(* IEC 61131-3 sources: crb-codesys/generation/scripts/repoeval/重型运输系统/core/FUN, 14 files *)

(* ---- percentCalc.st ---- *)
FUNCTION percentCalc : REAL
VAR_INPUT
	level		:INT;	//1->地轨	2->天轨
	idx			:INT;	//挡板索引编号
END_VAR
VAR
	c			:REAL;
	p			:REAL;
END_VAR

//伸出百分比计算
CASE level OF
	1:
		IF gDev.grd[idx].sensor.position < 3 THEN
			RETURN;
		END_IF
		c := gDev.grd[idx].sensor.position - gDev.grd[idx].sensor.retractVal;
		p := gDev.grd[idx].sensor.extendVal - gDev.grd[idx].sensor.retractVal;
		percentCalc := c * 100 / p;
	2:
		IF gDev.sky[idx].sensor.position < 3 THEN
			RETURN;
		END_IF
		c := gDev.sky[idx].sensor.position - gDev.sky[idx].sensor.retractVal;
		p := gDev.sky[idx].sensor.extendVal - gDev.sky[idx].sensor.retractVal;
		percentCalc := c * 100 / p;
END_CASE

(* ---- setButtonByDirect.st ---- *)
FUNCTION setButtonByDirect : BOOL
VAR_INPUT
	level		:INT;	//1->地轨	2->天轨
	idx			:INT;	//挡板索引编号
	direct		:TargetDirect;
END_VAR
VAR
END_VAR
//	本函数用于根据输入参数 操作UI界面的按钮变量
CASE level OF
	1:
		IF idx = 0 OR idx > 10 THEN		//参数校验
			RETURN;
		END_IF
		CASE direct OF
			TargetDirect.extend:
				gUI.grd[idx].btnStop := FALSE;
				gUI.grd[idx].btnExtend := TRUE;
				gUI.grd[idx].btnRetract := FALSE;
			TargetDirect.retract:
				gUI.grd[idx].btnStop := FALSE;
				gUI.grd[idx].btnExtend := FALSE;
				gUI.grd[idx].btnRetract := TRUE;
			TargetDirect.stop:
				gUI.grd[idx].btnStop := FALSE;
				gUI.grd[idx].btnExtend := FALSE;
				gUI.grd[idx].btnRetract := FALSE;
		END_CASE
	2:
		IF idx > 10 THEN		//参数校验
			RETURN;
		END_IF
		CASE direct OF
			TargetDirect.extend:
				gUI.sky[idx].btnStop := FALSE;
				gUI.sky[idx].btnExtend := TRUE;
				gUI.sky[idx].btnRetract := FALSE;
			TargetDirect.retract:
				gUI.sky[idx].btnStop := FALSE;
				gUI.sky[idx].btnExtend := FALSE;
				gUI.sky[idx].btnRetract := TRUE;
			TargetDirect.stop:
				gUI.sky[idx].btnStop := FALSE;
				gUI.sky[idx].btnExtend := FALSE;
				gUI.sky[idx].btnRetract := FALSE;
		END_CASE

END_CASE;

(* ---- updateDevStatus.st ---- *)
FUNCTION updateDevStatus : DevStatus
VAR_INPUT
	level		:INT;		//1->地轨	2->天轨
	idx			:INT;		//挡板索引编号
	errorVal	:REAL;		//误差范围
END_VAR
VAR
	extendVal	:REAL;		//伸出值
	retractVal	:REAL;		//缩回到位值
	nowVal		:REAL;		//当前值
	stat		:DevStatus;	//设备状态
END_VAR

(* 本函数用于根据设备的标定伸出/缩回值以及当前位置
** 判断该缸体是否处于伸出/缩回到位状态，如果到位更新参数
*)

stat := DevStatus.unknown;	//初始化状态量
CASE level OF
	1:
		extendVal := gDev.grd[idx].sensor.extendVal;
		retractVal := gDev.grd[idx].sensor.retractVal;
		nowVal := gDev.grd[idx].sensor.position;
		stat := gDev.grd[idx].state;
	2:
		extendVal := gDev.sky[idx].sensor.extendVal;
		retractVal := gDev.sky[idx].sensor.retractVal;
		nowVal := gDev.sky[idx].sensor.position;
		stat := gDev.sky[idx].state;
END_CASE

IF nowVal > 1 THEN
	IF nowVal < retractVal + errorVal THEN
		stat := DevStatus.retracted;
	ELSIF nowVal > extendVal - errorVal THEN
		stat := DevStatus.extended;
	ELSE
		IF stat <> DevStatus.runing THEN
			stat := DevStatus.error;
		END_IF
	END_IF
ELSE
	stat := DevStatus.unknown;
END_IF

CASE level OF
	1:
		gDev.grd[idx].state := stat;
	2:
		gDev.sky[idx].state := stat;
END_CASE

updateDevStatus := stat;

(* ---- BasePIDCtrl.st ---- *)
FUNCTION_BLOCK BasePIDCtrl
VAR_INPUT
	Act_Val 	:REAL;			//实际值
	Set_Val		:REAL;			//设定值
	Kp			:REAL;
	Ki			:REAL;
	Kd			:REAL;
	Y_MAX		:REAL;
	Y_MIN		:REAL;
	rCycle		:REAL;			//单位/s
	Reset		:BOOL;
END_VAR
VAR_OUTPUT
	Y			:REAL;
	LimitActive	:BOOL;
END_VAR
VAR
	fCycle			:REAL;
	CycleTime		:TIME ;
	Err				:REAL;    		//本次误差
	LastErr			:REAL;    		//上次误差
	KiErrSum		:REAL;			//积分累计误差
	KdErr			:REAL;			//微分误差
	Result			:REAL;			//计算结果
	Result_OUT		:REAL;		    //限制结果
	trig			:R_TRIG ;
	ton				:TON ;
END_VAR

IF  rCycle < 0.01 THEN  //10ms最小
	fCycle := 0.01;
ELSE
	fCycle := rCycle;
END_IF

CycleTime := REAL_TO_TIME (TIME_TO_REAL(T#1S) * fCycle);
ton (IN := NOT ton.Q ,PT := CycleTime ,Q =>);
trig (CLK := ton.Q  ,Q =>);

IF trig.Q THEN 			//PID计算
	Err := Set_Val - Act_Val;  //误差计算
	KiErrSum := KiErrSum + Err ;   //积分计算
	KdErr := Err -LastErr;    //微分计算
	LastErr := Err;
	(*IF ABS(Err) < 10 THEN		//误差较低时才开启积分
		KiErrSum := KiErrSum + Err ;   //积分计算
	END_IF*)
	Result :=  Kp * Err + Ki * KiErrSum + Kd * KdErr;
END_IF

IF Result > Y_MAX  THEN         //限幅度输出
	Result_OUT := Y_MAX ;
	LimitActive := TRUE ;
ELSIF Result < Y_MIN THEN
	Result_OUT := Y_MIN  ;
	LimitActive := TRUE ;
ELSE
	Result_OUT := Result ;
	LimitActive :=FALSE ;
END_IF
IF Reset THEN   //pid 不输出
	KiErrSum := 0;
	KdErr := 0;
	LastErr	:= 0;
	Y := 0;
ELSE
	Y := Result_OUT;
END_IF

(* ---- CommandExecutor.st ---- *)
FUNCTION_BLOCK CommandExecutor
VAR_INPUT
	level		:INT;			//1->地轨	2->天轨
	idx			:INT;			//挡板索引编号
	percent		:REAL;			//比例阀百分比 传入-100~+100
END_VAR
VAR_OUTPUT
END_VAR
VAR
END_VAR

IF percent > 0 THEN
	CASE level OF
		1:
			gController.grd[idx].extendPercent := REAL_TO_WORD(percent * 65535 / 100);
			gController.grd[idx].retractPercent := 0;
		2:
			gController.sky[idx].extendPercent := REAL_TO_WORD(percent * 65535 / 100);
			gController.sky[idx].retractPercent := 0;
	END_CASE
ELSE
	CASE level OF
		1:
			gController.grd[idx].extendPercent := 0;
			gController.grd[idx].retractPercent := REAL_TO_WORD(ABS(percent) * 65535 / 100);
		2:
			gController.sky[idx].extendPercent := 0;
			gController.sky[idx].retractPercent := REAL_TO_WORD(ABS(percent) * 65535 / 100);
	END_CASE
END_IF

(* ---- CommandExecutor0.st ---- *)
FUNCTION_BLOCK CommandExecutor0
VAR_INPUT
	level		:INT;			//1->地轨	2->天轨
	idx			:INT;			//挡板索引编号
	direct		:TargetDirect;	//方向
	percent		:REAL;			//比例阀百分比 传入0-100
END_VAR
VAR_OUTPUT
END_VAR
VAR
END_VAR

CASE direct OF
	TargetDirect.extend:
		CASE level OF
			1:
				gController.grd[idx].extendPercent := REAL_TO_WORD(percent * 65535 / 100);
				gController.grd[idx].retractPercent := 0;
			2:
				gController.sky[idx].extendPercent := REAL_TO_WORD(percent * 65535 / 100);
				gController.sky[idx].retractPercent := 0;
		END_CASE
	TargetDirect.retract:
		CASE level OF
			1:
				gController.grd[idx].extendPercent := 0;
				gController.grd[idx].retractPercent := REAL_TO_WORD(percent * 65535 / 100);
			2:
				gController.sky[idx].extendPercent := 0;
				gController.sky[idx].retractPercent := REAL_TO_WORD(percent * 65535 / 100);
		END_CASE
	TargetDirect.stop:
		CASE level OF
			1:
				gController.grd[idx].extendPercent := 0;
				gController.grd[idx].retractPercent := 0;
			2:
				gController.sky[idx].extendPercent := 0;
				gController.sky[idx].retractPercent := 0;
		END_CASE

	ELSE
		CASE level OF
			1:
				gController.grd[idx].extendPercent := 0;
				gController.grd[idx].retractPercent := 0;
			2:
				gController.sky[idx].extendPercent := 0;
				gController.sky[idx].retractPercent := 0;
		END_CASE

END_CASE

(* ---- fileSave.st ---- *)
FUNCTION_BLOCK fileSave
VAR_INPUT
	filePath 	:STRING;
	intervalt	:INT;
END_VAR
VAR
	lineCount	: INT;
	fileHandle  : DWORD;
	fileName	: STRING;
END_VAR
VAR_OUTPUT
END_VAR

(* ---- fileSave_close.st ---- *)
FUNCTION_BLOCK fileSave
VAR_INPUT
	filePath 	:STRING;
	intervalt	:INT;
END_VAR
VAR
	lineCount	: INT;
	fileHandle  : DWORD;
	fileName	: STRING;
END_VAR
VAR_OUTPUT
END_VAR

IF fileHandle <> 0 THEN
	SysFileClose(hFile := fileHandle);
	fileHandle := 0;
END_IF

(* ---- fileSave_createDir.st ---- *)
FUNCTION_BLOCK fileSave
VAR_INPUT
	filePath 	:STRING;
	devName		: STRING ;
	intervalt	:INT;
END_VAR
VAR
	lineCount	: INT;
	fileHandle  : DWORD;
	fileName	: STRING;
	filePath1	:STRING;
END_VAR
VAR_OUTPUT
END_VAR

filePath1 := FilePath;
filePath1 := concat(filePath1,'/');
filePath1 := concat(filePath1,devName);
SysDirCreate2(filePath1, TRUE);

(* ---- fileSave_new.st ---- *)
FUNCTION_BLOCK fileSave
VAR_INPUT
	filePath 	:STRING;
	intervalt	:INT;
	devName		: STRING ;
END_VAR
VAR
	lineCount	: INT;
	fileHandle  : DWORD;
	fileName	: STRING;
	fileHandle0 : DWORD;
	datetime	: DATE_AND_TIME;
	UdIntms 	: UDINT;
	UdMsOffset  : UDINT;
	DTimer_Str  : STRING;
	uiYear 		: UINT;
    uiMonth 	: UINT;
    uiDay 		: UINT;
    uiHour 		: UINT;
    uiMinute 	: UINT;
    uiSecond 	: UINT;
	uiMsSecond	: UINT;

	S_Time64		:  SysTime64;
	STT			:  CurTimeEx;
	S_Time			:  SystemTimeDate;
	Time_Str		:  STRING;
	F_err		: DWORD;
	F_HANDL		: DWORD;
END_VAR
VAR_OUTPUT
END_VAR

	STT(SystemTime:= S_Time64, TimeDate:= S_Time);
	Time_Str :='';
	Time_Str := concat(Time_Str,UINT_TO_STRING(S_Time.Year));
	Time_Str := concat(Time_Str,'-');
	Time_Str := concat(Time_Str,UINT_TO_STRING(S_Time.Month));
	Time_Str := concat(Time_Str,'-');
	Time_Str := concat(Time_Str,UINT_TO_STRING(S_Time.Day));
	Time_Str := concat(Time_Str,'_');
	Time_Str := concat(Time_Str,UINT_TO_STRING(S_Time.Hour));
	Time_Str := concat(Time_Str,'-');
	Time_Str := concat(Time_Str,UINT_TO_STRING(S_Time.Minute));
	Time_Str := concat(Time_Str,'-');
	Time_Str := concat(Time_Str,UINT_TO_STRING(S_Time.Second));
	Time_Str := concat(Time_Str,'_');
	Time_Str := concat(Time_Str,UINT_TO_STRING(S_Time.Milliseconds));

	fileName := FilePath;
	fileName := concat(fileName,'/');
	fileName := concat(fileName,devName);

	fileName := concat(fileName,'/');
	fileName := concat(fileName,devName);
	fileName := concat(fileName,'-');
	fileName := concat(fileName,Time_Str);
    fileName := concat(fileName,'.txt');

	fileHandle := SysFileOpen(szFile:= fileName, am:=ACCESS_MODE.AM_WRITE, pResult:= ADR(F_err));
	lineCount := -1;
	//fileHandle := SysFileOpen(szFile:= fileName, am:=ACCESS_MODE.AM_APPEND, pResult:= ADR(F_err));

(* ---- fileSave_write.st ---- *)
FUNCTION_BLOCK fileSave
VAR_INPUT
	filePath 	:STRING;
	intervalt	:INT;
	positionInt 	:INT;
	speedInt 		:INT;
	stateInt		:INT;
END_VAR
VAR
	lineCount	: INT;
	fileHandle  : DWORD;
	fileName	: STRING;
	data		: STRING;
	F_err		: DWORD;
	tempInt		: INT;
END_VAR
VAR_OUTPUT
END_VAR

IF fileHandle <> 0 THEN
	lineCount := lineCount + 1;
	tempInt	:= lineCount * intervalt;
	data := INT_TO_STRING(lineCount);
	data := concat(data,'$T$T');
	data := concat(data, INT_TO_STRING(tempInt));
	IF tempInt < 1000 THEN
		data := concat(data,'$T');
	END_IF
	data := concat(data,'$T$T');
	data := concat(data,INT_TO_STRING(positionInt));
	data := concat(data,'$T');
	data := concat(data,INT_TO_STRING(speedInt));
	data := concat(data,'$T');
	data := concat(data,INT_TO_STRING(stateInt));
	data := concat(data,'$R');

	SysFileWrite(hFile:=fileHandle , pbyBuffer:= ADR(data) , ulSize:= DINT_TO_DWORD(SysStrLen(data)) , pResult:= ADR(F_err));		// 写入数据

END_IF

(* ---- grdPosCtrl.st ---- *)
FUNCTION_BLOCK grdPosCtrl
VAR_INPUT
	idx			:INT;			//挡板索引编号
	isReset		:BOOL;
	cycTimer	:REAL;
END_VAR

VAR_OUTPUT
	res		:REAL;
END_VAR
VAR
	posPid		:BasePIDCtrl;
	spdPid		:BasePIDCtrl;
	setSpeed	:REAL;
	overBase	:REAL;
	out			:REAL;
	controller	:DevPid;
END_VAR

controller := gDev.grd[idx].ctrl;
posPid(
	Act_Val:= gDev.grd[idx].sensor.position,
	Set_Val:= controller.pos.Set_Point,
	Kp:= controller.pos.Kp,
	Ki:= controller.pos.Ki,
	Kd:= controller.pos.Kd,
	Y_MAX:= controller.pos.Max_Val,     //最大速度
	Y_MIN:= -controller.pos.Max_Val,    //水平运动正反一致
	rCycle:= 0.1,   //位置计算周期 100ms
	Reset:= isReset,
	Y => controller.pos.OUT,
	LimitActive=> );

IF ABS(posPid.Y - setSpeed) > (cycTimer * controller.pos.Max_ACC) THEN
	IF posPid.Y > setSpeed THEN
		setSpeed := setSpeed + (cycTimer * controller.pos.Max_ACC);
	ELSE
		setSpeed := setSpeed - (cycTimer * controller.pos.Max_ACC);
	END_IF
ELSE
	setSpeed := posPid.Y;
END_IF

controller.spd.Set_Point := setSpeed;

IF setSpeed > 0 THEN
	overBase := setSpeed * controller.ff.pstKv + controller.ff.pstThreshold;
ELSE
	overBase := setSpeed * controller.ff.negKv - controller.ff.negThreshold;
END_IF

spdPid(
	Act_Val:= gDev.grd[idx].sensor.speed,
	Set_Val:= controller.spd.Set_Point,
	Kp:= controller.spd.Kp,
	Ki:= controller.spd.Ki,
	Kd:= controller.spd.Kd,
	Y_MAX:= controller.spd.Max_Val,     //最大速度
	Y_MIN:= -controller.spd.Max_Val,    //水平运动正反一致
	rCycle:= 0.02,   //位置计算周期 100ms
	Reset:= isReset,
	Y=> ,
	LimitActive=> );

out := spdPid.Y + overBase;
IF out > controller.spd.Max_Val THEN
	out := controller.spd.Max_Val;
END_IF
IF out < -controller.spd.Max_Val THEN
	out := -controller.spd.Max_Val;
END_IF
IF isReset	THEN out := 0;	END_IF
controller.spd.OUT := out;
gDev.grd[idx].ctrl := controller;
res := out;

(* ---- skyPosCtrl.st ---- *)
FUNCTION_BLOCK skyPosCtrl
VAR_INPUT
	idx			:INT;			//挡板索引编号
	isReset		:BOOL;
	cycTimer	:REAL;
END_VAR

VAR_OUTPUT
	res		:REAL;
END_VAR
VAR
	posPid		:BasePIDCtrl;
	spdPid		:BasePIDCtrl;
	setSpeed	:REAL;
	overBase	:REAL;
	out			:REAL;
	//fb_Val		:REAL;
	controller	:DevPid;
END_VAR

controller := gDev.sky[idx].ctrl;
posPid(
	Act_Val:= gDev.sky[idx].sensor.position,
	Set_Val:= controller.pos.Set_Point,
	Kp:= controller.pos.Kp,
	Ki:= controller.pos.Ki,
	Kd:= controller.pos.Kd,
	Y_MAX:= controller.pos.Max_Val,     //最大速度
	Y_MIN:= -controller.pos.Max_Val,    //水平运动正反一致
	rCycle:= 0.05,   //位置计算周期 100ms
	Reset:= isReset,
	Y => controller.pos.OUT,
	LimitActive=> );

IF ABS(posPid.Y - setSpeed) > (cycTimer * controller.pos.Max_ACC) THEN
	IF posPid.Y > setSpeed THEN
		setSpeed := setSpeed + (cycTimer * controller.pos.Max_ACC);
	ELSE
		setSpeed := setSpeed - (cycTimer * controller.pos.Max_ACC);
	END_IF
ELSE
	setSpeed := posPid.Y;
END_IF

controller.spd.Set_Point := setSpeed;

IF setSpeed > 0 THEN
	overBase := setSpeed * controller.ff.pstKv + controller.ff.pstThreshold;
END_IF
IF setSpeed < 0 THEN
	overBase := setSpeed * controller.ff.negKv - controller.ff.negThreshold;
END_IF

spdPid(
	Act_Val:= gDev.sky[idx].sensor.speed,
	Set_Val:= controller.spd.Set_Point,
	Kp:= controller.spd.Kp,
	Ki:= controller.spd.Ki,
	Kd:= controller.spd.Kd,
	Y_MAX:= controller.spd.Max_Val,     //最大速度
	Y_MIN:= -controller.spd.Max_Val,    //水平运动正反一致
	rCycle:= 0.02,   //位置计算周期 100ms
	Reset:= isReset,
	Y=> ,
	LimitActive=> );

out := spdPid.Y + overBase;

IF out > controller.spd.Max_Val THEN
	out := controller.spd.Max_Val;
END_IF
IF out < -controller.spd.Max_Val THEN
	out := -controller.spd.Max_Val;
END_IF
IF isReset	THEN out := 0;	END_IF
controller.spd.OUT := out;
gDev.sky[idx].ctrl := controller;
res := out;

(* ---- tcpUpload_send.st ---- *)
FUNCTION_BLOCK tcpUpload
VAR_INPUT
	InetAddress		:STRING;
	port			:UINT;
	dataLength		:__XINT;
	sendBuf 		:ARRAY[1..1024]OF BYTE;
END_VAR
VAR_OUTPUT
END_VAR
VAR
	tcpConnector	:TCP.Connector;
	tcpStream		:TCP.Stream;
	pointerStream	:POINTER TO TCP.Stream;
	sizeData		:__XINT;

	tcpState		:UINT:=0;
	tcpCount		:UINT:=0;

	netState		:INT;
END_VAR

tcpCount := tcpCount + 1;
CASE tcpState OF

	0:			//connet server
		tcpConnector.Connect(sIPAddress:= InetAddress,uiPort:= port,pStream => pointerStream);
		IF pointerStream<>0 THEN
			tcpState :=1;
		ELSE
			tcpState :=2;
		END_IF

	1:
		netState := pointerStream^.Send(ADR(sendBuf),dataLength,diSent=>sizeData);
		IF netState <> 0 THEN
			tcpState := 2;
		END_IF

	2:		 	//断开连接
	    tcpConnector.Disconnect();
		tcpState := 0;

END_CASE
